// TIA Portal V17 export
// export: Created 2025-05-06T14:44:46.1175146Z, ExportSetting WithDefaults, DisplayName Totally Integrated Automation Portal, DisplayVersion V17 Update 8, DisplayName TIA Portal Openness, DisplayVersion V17 Update 8, DisplayName TIA Portal Version Control Interface, DisplayVersion V17, DisplayName SINAMICS Startdrive Advanced, DisplayVersion V17 SP2, DisplayName SINAMICS Startdrive G110M, G120, G120C, G120D, G120P, G115D, DisplayVersion V17 SP2, DisplayName SINAMICS Startdrive G130, G150, S120, S150, SINAMICS MV, S210, DisplayVersion V17 SP2, DisplayName STEP 7 Professional, DisplayVersion V17 Update 8, DisplayName SINUMERIK ONE STEP 7 Toolbox, DisplayVersion V17 Update 12, DisplayName SINUMERIK 840D sl STEP 7 Toolbox, DisplayVersion V17 Update 12, DisplayName STEP 7 Safety, DisplayVersion V17 Update 6, DisplayName WinCC Advanced, DisplayVersion V17 Update 8
DATA_BLOCK "DB7272_HOPPER_1_UNIT_02"   // DB7272
{ DB_Accessible_From_OPC_UA := 'FALSE' }
VERSION : 0.1
// stored: AutoNumber false, DBAccessibleFromOPCUA false, DBAccessibleFromWebserver true, InstanceOfName FB7240_VARIABLES_PLC_HMI_HOPPERS, InstanceOfType FB
"FB7240_VARIABLES_PLC_HMI_HOPPERS"
   // VAR_INPUT
   //    STIRRER_SPEED_ACTUAL : DInt;
   //    STIRRER_SPEED_CONS : DInt;
   //    STIRRER_STARTED : Bool;
   //    UPPER_JACKET_ACTUAL : Real;
   //    UPPER_JACKET_CONS : Real;
   //    UPPER_JACKET_STARTED : Bool;
   //    LOWER_JACKET_ACTUAL : Real;
   //    LOWER_JACKET_CONS : Real;
   //    LOWER_JACKET_STARTED : Bool;
   //    HOPPER_COVER_ACTUAL : Real;
   //    HOPPER_COVER_CONS : Real;
   //    HOPPER_COVER_STARTED : Bool;
   //    FEEDING_COVER_ACTUAL : Real;
   //    FEEDER_DISK_PRESS_ACTUAL : Real;
   //    POWDER_WEIGHT_ACTUAL : Real;
   //    PRESSURIZE_VALVE_OPEN : Bool;
   //    PRESSURIZE_VALVE_CLOSED : Bool;
   //    RELIEVE_VALVE_OPEN : Bool;
   //    RELIEVE_VALVE_CLOSED : Bool;
   //    TRANSFER_VALVE_OPEN : Bool;
   //    TRANSFER_VALVE_CLOSED : Bool;
   //    LOAD_FEEDER_TIME_SEQUENCE_STARTED : Bool;
   //    LOAD_FEEDER_TIME_SEQUENCE_STOPPED : Bool;
   //    LOAD_FEEDER_WEIGHT_SEQUENCE_STARTED : Bool;
   //    LOAD_FEEDER_WEIGHT_SEQUENCE_STOPPED : Bool;
   //    HOPPER_POWDER_LOW_LEVEL_SIGNAL_ON : Bool;
   //    HOPPER_POWDER_HIGH_LEVEL_SIGNAL_ON : Bool;
   //    FEEDER_CURRENT_VALUE : Real;
   // END_VAR
   // VAR_OUTPUT
   //    STIRRER_SPEED_SETPOINT : DInt;
   //    UPPER_JACKET_SETPOINT : Real;
   //    LOWER_JACKET_SETPOINT : Real;
   //    HOPPER_COVER_SETPOINT : Real;
   //    LOAD_FEED_SEQ_HIGH_LIMIT_CURRENT : UInt;
   //    LOAD_FEED_SEQ_LOW_LIMIT_CURRENT : UInt;
   //    LOAD_FEED_TIME_SEQ_INCREMENT_PRESS_VALUE : Real;
   //    LOAD_FEED_TIME_SEQ_SET_TIME_VALUE : UDInt;
   //    LOAD_FEED_WEIGHT_SEQ_INCREMENT_PRESS_VALUE : Real;
   //    LOAD_FEED_WEIGHT_SEQ_SET_WEIGHT_VALUE : Real;
   // END_VAR
   // VAR_IN_OUT
   //    HOPPER_LINE_IN_OUT : "UDT_Hopper Line";
   // END_VAR
BEGIN
END_DATA_BLOCK
